// TwinCAT 3 PLC project SetDecimal
// ProgramVersion: 3.1.4024.0
// libraries:
//   Tc2_Standard, * (Beckhoff Automation GmbH)
//   Tc2_System, * (Beckhoff Automation GmbH)
//   Tc3_Module, * (Beckhoff Automation GmbH)
// project tree:
//   GVLs/ GVL.TcGVL
//   / PlcTask.TcTTO
//   POUs/ F_ROUND_REAL_GLOBAL.TcPOU, MAIN.TcPOU, F_ROUND_REAL.TcPOU
// real-time tasks:
//   TASK PlcTask: cycle T#10ms, priority 20, ADS port 350

CONFIGURATION SetDecimal
    RESOURCE PLC ON TwinCAT3
        TASK PlcTask(INTERVAL := T#10ms, PRIORITY := 20);
        PROGRAM MAIN WITH PlcTask : MAIN;
    END_RESOURCE
END_CONFIGURATION

// ---- GVLs/GVL.TcGVL
{attribute 'qualified_only'}
VAR_GLOBAL
	rRoundedValue 	: ARRAY[1..6] OF REAL;
	rRawValue		: ARRAY[1..6] OF REAL := [1.111,2.222,3.666,4.888,5.555,6.159];
END_VAR

// ---- POUs/MAIN.TcPOU
PROGRAM MAIN
VAR
	rRoundedValue 	: ARRAY[1..6] OF REAL;
	rRawValue		: ARRAY[1..6] OF REAL := [1.111,2.222,3.666,4.888,5.555,6.159];
END_VAR

rRoundedValue := F_ROUND_REAL(rRawValue, 1);
GVL.rRoundedValue := F_ROUND_REAL_GLOBAL(1);

END_PROGRAM

// ---- POUs/F_ROUND_REAL.TcPOU
FUNCTION F_ROUND_REAL : REAL
VAR_INPUT
  rInput 			: REAL;
  iDecimalPlaces 	: INT;
END_VAR
VAR
  rOutput 			: real;
  rLeftPart 		: REAL;
  Value				: dint;
END_VAR


rOutput := rInput * EXPT(10,iDecimalPlaces);
//rLeftPart := rOutput - TRUNC(rOutput);

//IF rLeftPart >= 0.5 THEN
//  rOutput := rOutput + 1;
//ElSIF rLeftPart <= -0.5 THEN
//  rOutput := rOutput - 1;
//ELSE
//  rOutput := rOutput;
//END_IF

Value := REAL_TO_DINT(rOutput);
rOutput := Value / EXPT(10,iDecimalPlaces);
F_ROUND_REAL := rOutput;

END_FUNCTION

// ---- POUs/F_ROUND_REAL_GLOBAL.TcPOU
FUNCTION F_ROUND_REAL_GLOBAL : ARRAY[1..6] OF REAL
VAR_INPUT
  iDecimalPlaces 	: INT;
END_VAR
VAR
  rOutput 			: ARRAY[1..6] OF REAL;
  Value				: ARRAY[1..6] OF DINT;
  X					: int;
END_VAR

FOR X := 1 TO 6 BY 1 DO
	rOutput[X] := LREAL_TO_REAL(GVL.rRawValue[X] * EXPT(10,iDecimalPlaces));
	Value[X] := REAL_TO_DINT(rOutput[X]);
	rOutput[X] := LREAL_to_real(Value[X] / EXPT(10,iDecimalPlaces));
END_FOR

F_ROUND_REAL_GLOBAL := rOutput;

END_FUNCTION
